Omron CX-Programmer project НовыйПроект (CX-Programmer 9.54)

# PLC НовыйПЛК1: CP1L L

## Program НоваяЗадача1 (cyclic task 0)

### Section Сегмент1

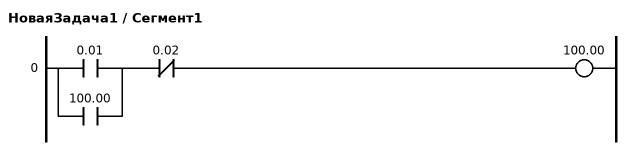
; rung 0
LD 0.01
OR 100.00
ANDNOT 0.02
OUT 100.00

### Section END
; rung 0
END(001)